{attribute 'Tc2GvlVarNames'}
VAR_GLOBAL CONSTANT
(*************************************************************************************************)
(*  FILENAME:    DEFINTIONS.EXP                                                                  *)
(*  PROJECT:     CALMAR PUPLC                                                                    *)
(*  COPYRIGHT:   All rights reserved (c) Wifag//Polytype, Fribourg/Switzerland (2016)            *)
(*  ENVIRONMENT: TwinCAT PLC                                                                     *)
(*  VERSION:     <version>                                                                       *)
(*************************************************************************************************)
(*  DESCRIPTION:                                                                   <description> *)
(*    Global variable constant.                                                                  *)
(*                                                                                </description> *)
(*************************************************************************************************)

  aC_NAME_PROJECT               : STRING   := 'DP-ST-1026-WEU2';
  aC_NAME_PRODUCT               : STRING   := 'WEU';
  aC_VERSION_PRODUCT            : STRING   := '01.000.000';
  iC_VERSION_PRODUCT            : INT      := 010000;

  sC_AMSNETID_LOCALHOST         : STRING   := '';                   (* AMS_NET_ID of Localhost *)
  sC_AMSNETID_IO                : STRING   := '172.21.10.11.2.1';   (* AMS_NET_ID of IO *)

  aC_WifagDataPath              : STRING[255] := 'C:\ProgramData\WifagPolytype\';     (*Path of Wifag ProgramData*)
  aC_PlcSubPath                 : STRING[255] := 'PrintUnitPlc\02_Plc\';              (*Sub path to 02_PLC*)
  aC_RecipeSubPath              : STRING[255] := 'Recipe\';                           (*Sub path to recipe*)

  aC_PlcConfigPath              : STRING   := 'C:\ProgramData\WifagPolytype\WEUPrintUnitPlc\';   (*Plc config / report data path*)
  aC_PlcFlashFileSubPath        : STRING   := '03_Flash\';     (*firmware file sub-directory*)
  aC_PlcWaveformFileSubPath     : STRING   := '04_Waveform\';  (*waveform file sub-directory*)
  aC_PlcMaskFileSubPath         : STRING   := '05_Mask\';      (*stiching mask file sub-directory*)
  aC_PlcMapFileSubPath          : STRING   := '06_Map\';       (*correction map file sub-directory*)
  aC_PlcRecipeSubPath           : STRING   := '02_Plc\Recipe\';(*recipe file sub-directory*)  
  aC_PlcBlockIdSubPath          : STRING   := '02_Plc\BlockId\';(*blockId file sub-directory*)
  aC_PlcAlarmDbSubPath          : STRING   := '02_Plc\AlarmDb\';(*alarm db file sub-directory*)
  
  aC_PlcProjectCfgPath          : T_MaxString := 'C:\ProgramData\WifagPolytype\WEUPrintUnitPlc\02_Plc\DPST-1026-WEU 2 Demo\WEU2\PlcProject\Configuration\';
  
  
  iG_PC_ADDRESS                 : ARRAY[1..32] OF UINT := [1050,
                                                           1051,
                                                           1052,
                                                           1053,
                                                           1054,
                                                           1055,
                                                           1056,
                                                           1057,
                                                           1058,
                                                           1059];

END_VAR

(* stored: Version 1.1.0.1, ProductVersion 3.1.4024.11
   GVL Definitions: Id {b1e2f023-9af0-4663-a1f8-d114142fdd31} *)
